Fanuc TP program (LS listing): UP025.LS

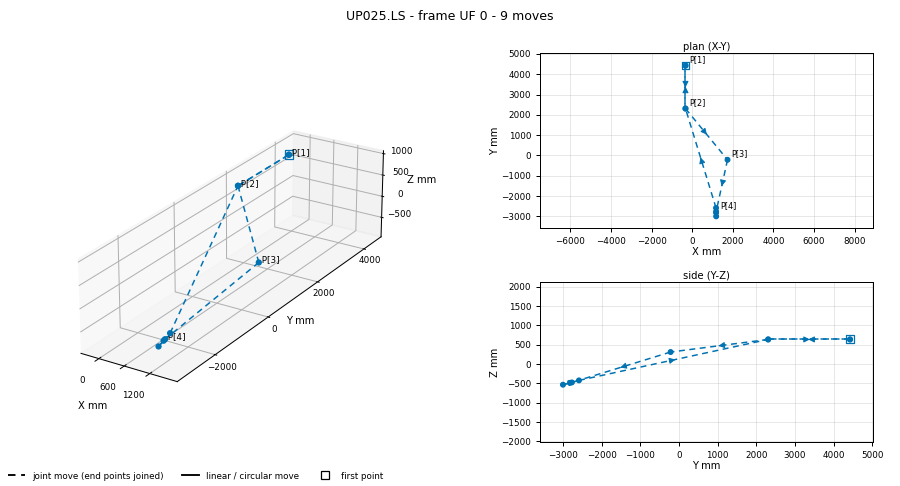
[picture p0: tool path of UP025.LS in frame UF 0, 9 of 9 moves have a stored position in this frame; points joined in program order, loops and branches not executed]
/PROG  UP025
/ATTR
OWNER		= MNEDITOR;
COMMENT		= "Int. 1680 Pos. 1";
PROG_SIZE	= 4392;
CREATE		= DATE 23-07-11  TIME 01:05:50;
MODIFIED	= DATE 24-07-27  TIME 15:01:24;
FILE_NAME	= UP005;
VERSION		= 0;
LINE_COUNT	= 18;
MEMORY_SIZE	= 7892;
PROTECT		= READ_WRITE;
TCD:  STACK_SIZE	= 500,
      TASK_PRIORITY	= 50,
      TIME_SLICE	= 0,
      BUSY_LAMP_OFF	= 0,
      ABORT_REQUEST	= 0,
      PAUSE_REQUEST	= 0;
DEFAULT_GROUP	= 1,1,1,1,*;
CONTROL_CODE	= 00000000 00000000;
/APPL
/MN
   1:  UFRAME_NUM=0 ;
   2:  UTOOL_NUM=1 ;
   3:  PAYLOAD[1] ;
   4:  !Apagar Perfil Lib. 77 vs ST1680 ;
   5:J P[1] 100% CNT0 ACC100 TB   0.00sec,P-SPS    ;
      1:  TC_ONLINE (ON) ;
      2:  DO[23]=OFF ;
      3:  TIMER[6]=RESET ;
      4:  TIMER[6]=START ;
      5:  CALL MAKRO050    ;
      6:  !Lib. de Herramientas ;
      7:  DO[80]=ON ;
      8:  DO[78]=OFF ;
      9:  DO[77]=ON ;
     10:  DO[75]=OFF ;
     11:  DO[74]=ON ;
     12:  DO[72]=OFF ;
     13:  !Lib. de Anticolisiones ;
     14:  DO[43]=ON ;
     15:  DO[44]=ON ;
     16:  !Apagar Pos. Base ;
     17:  DO[15]=OFF ;
     18:  !Robot en Trayectoria ;
     19:  DO[16]=ON ;
     20:  WAIT (!DI[61] AND DI[62] AND DI[77] AND M[2])    ;
     21:  DO[77]=OFF ;
     22:  WAIT (DI[23])    ;
     23:  DO[23]=ON ;
     24:  TC_ONLINE (!DI[61] AND DI[62] AND DI[77] AND M[2] AND M[30] AND M[31] AND M[33]) ;
       ------ ;
   6:J P[2] 100% CNT100 ACC100 TB   0.00sec,P-SPS    ;
      1:  TC_ONLINE (!DI[61] AND DI[62] AND DI[77] AND M[2] AND M[30] AND M[31] AND M[33]) ;
       ------ ;
   7:J P[3] 100% CNT100 ACC100 TB   0.00sec,P-SPS    ;
      1:  TC_ONLINE (!DI[61] AND DI[62] AND DI[77] AND M[2] AND M[30] AND M[31] AND M[33]) ;
       ------ ;
   8:J P[4] 100% CNT0 ACC100 TB    .10sec,P-SPS    ;
      1:  TC_ONLINE (ON) ;
      2:  DO[23]=OFF ;
      3:  F[2]=(ON) ;
      4:  CALL MAKRO343    ;
      5:  WAIT (M[34])    ;
      6:  WAIT (DI[23])    ;
      7:  DO[23]=ON ;
      8:  TC_ONLINE (DI[77] AND M[30] AND M[31] AND M[34]) ;
       ------ ;
   9:  !En Posicion ST1680-1 ;
  10:  !Tomar Pieza en ST1680-1 ;
  11:  !Fin de Trabajo 3 ;
  12:L P[5] 200mm/sec CNT0 ACC100 TB   0.00sec,P-SPS    ;
      1:  TC_ONLINE (ON) ;
      2:  DO[23]=OFF ;
      3:  DO[75]=ON ;
      4:  WAIT (M[1])    ;
      5:  F[2]=(ON) ;
      6:  CALL MAKRO342    ;
      7:  CALL MAKRO340    ;
      8:  WAIT (M[33])    ;
      9:  F[1]=(ON) ;
     10:  CALL MAKRO343    ;
     11:  WAIT (M[32])    ;
     12:  CALL MAKRO003    ;
     13:  GO[21]=2 ;
     14:  WAIT (DI[77])    ;
     15:  DO[75]=OFF ;
     16:  WAIT (DI[23])    ;
     17:  DO[23]=ON ;
     18:  TC_ONLINE (DI[77] AND M[30] AND M[32] AND M[33]) ;
       ------ ;
  13:  PAYLOAD[2] ;
  14:L P[6] 300mm/sec CNT0 ACC100 TB    .10sec,P-SPS    ;
      1:  TC_ONLINE (ON) ;
      2:  DO[23]=OFF ;
      3:  WAIT (DI[61] AND !DI[62])    ;
      4:  WAIT (DI[23])    ;
      5:  DO[23]=ON ;
      6:  TC_ONLINE (DI[61] AND !DI[62] AND DI[77] AND M[1] AND M[30] AND M[32] AND M[33]) ;
       ------ ;
  15:J P[7] 90% CNT100 ACC50 TB   0.00sec,P-SPS    ;
      1:  TC_ONLINE (DI[61] AND !DI[62] AND DI[77] AND M[1] AND M[30] AND M[32] AND M[33]) ;
       ------ ;
  16:J P[8] 90% CNT100 ACC75 TB   0.00sec,P-SPS    ;
      1:  TC_ONLINE (DI[61] AND !DI[62] AND DI[77] AND M[1] AND M[30] AND M[32] AND M[33]) ;
       ------ ;
  17:  !Encender Perfil Lib 77 vs ST1680 ;
  18:J P[9] 90% CNT0 ACC50 TB    .10sec,P-SPS    ;
      1:  TC_ONLINE (ON) ;
      2:  DO[23]=OFF ;
      3:  TIMER[6]=STOP ;
      4:  DO[77]=ON ;
      5:  WAIT (DI[23])    ;
      6:  DO[23]=ON ;
      7:  TC_ONLINE (M[1] AND M[30] AND M[32] AND M[33]) ;
       ------ ;
/POS
P[1]{
   GP1:
	UF : 0, UT : 1,		CONFIG : 'F U T, 0, 0, 0',
	X =  -332.978  mm,	Y =  4426.811  mm,	Z =   636.000  mm,
	W =    91.999 deg,	P =      .001 deg,	R =  -180.000 deg,
	E1=  2500.000  mm
   GP2:
	UF : 0, UT : 1,
	J1=     0.000  mm
   GP3:
	UF : 0, UT : 1,
	J1=     0.000  mm
   GP4:
	UF : 0, UT : 1,
	J1=     0.000  mm
};
P[2]{
   GP1:
	UF : 0, UT : 1,		CONFIG : 'F U T, 0, 0, 0',
	X =  -332.978  mm,	Y =  2308.572  mm,	Z =   636.000  mm,
	W =    91.999 deg,	P =     0.000 deg,	R =   180.000 deg,
	E1=   381.761  mm
   GP2:
	UF : 0, UT : 1,
	J1=     0.000  mm
   GP3:
	UF : 0, UT : 1,
	J1=     0.000  mm
   GP4:
	UF : 0, UT : 1,
	J1=     0.000  mm
};
P[3]{
   GP1:
	UF : 0, UT : 1,		CONFIG : 'F U T, 0, 0, 0',
	X =  1737.304  mm,	Y =  -214.852  mm,	Z =   310.171  mm,
	W =   -92.297 deg,	P =    29.499 deg,	R =   -87.049 deg,
	E1=   -31.039  mm
   GP2:
	UF : 0, UT : 1,
	J1=     0.000  mm
   GP3:
	UF : 0, UT : 1,
	J1=     0.000  mm
   GP4:
	UF : 0, UT : 1,
	J1=     0.000  mm
};
P[4]{
   GP1:
	UF : 0, UT : 1,		CONFIG : 'F U T, 0, 0, 0',
	X =  1175.296  mm,	Y = -2769.815  mm,	Z =  -476.333  mm,
	W =   -88.686 deg,	P =    14.319 deg,	R =   -89.512 deg,
	E1=   -67.734  mm
   GP2:
	UF : 0, UT : 1,
	J1=     0.000  mm
   GP3:
	UF : 0, UT : 1,
	J1=     0.000  mm
   GP4:
	UF : 0, UT : 1,
	J1=     0.000  mm
};
P[5]{
   GP1:
	UF : 0, UT : 1,		CONFIG : 'F U T, 0, 0, 0',
	X =  1177.251  mm,	Y = -2999.679  mm,	Z =  -535.012  mm,
	W =   -88.686 deg,	P =    14.320 deg,	R =   -89.512 deg,
	E1=   -67.734  mm
   GP2:
	UF : 0, UT : 1,
	J1=     0.000  mm
   GP3:
	UF : 0, UT : 1,
	J1=     0.000  mm
   GP4:
	UF : 0, UT : 1,
	J1=     0.000  mm
};
P[6]{
   GP1:
	UF : 0, UT : 1,		CONFIG : 'F U T, 0, 0, 0',
	X =  1174.699  mm,	Y = -2819.354  mm,	Z =  -487.291  mm,
	W =   -88.458 deg,	P =    14.512 deg,	R =   -89.509 deg,
	E1=   -67.734  mm
   GP2:
	UF : 0, UT : 1,
	J1=     0.000  mm
   GP3:
	UF : 0, UT : 1,
	J1=     0.000  mm
   GP4:
	UF : 0, UT : 1,
	J1=     0.000  mm
};
P[7]{
   GP1:
	UF : 0, UT : 1,		CONFIG : 'F U T, 0, 0, 0',
	X =  1172.046  mm,	Y = -2585.848  mm,	Z =  -423.241  mm,
	W =   -88.895 deg,	P =    14.619 deg,	R =   -89.503 deg,
	E1=   -67.735  mm
   GP2:
	UF : 0, UT : 1,
	J1=     0.000  mm
   GP3:
	UF : 0, UT : 1,
	J1=     0.000  mm
   GP4:
	UF : 0, UT : 1,
	J1=     0.000  mm
};
P[8]{
   GP1:
	UF : 0, UT : 1,		CONFIG : 'F U T, 0, 0, 0',
	X =  -332.978  mm,	Y =  2308.572  mm,	Z =   636.000  mm,
	W =    91.999 deg,	P =     0.000 deg,	R =  -180.000 deg,
	E1=   381.761  mm
   GP2:
	UF : 0, UT : 1,
	J1=     0.000  mm
   GP3:
	UF : 0, UT : 1,
	J1=     0.000  mm
   GP4:
	UF : 0, UT : 1,
	J1=     0.000  mm
};
P[9]{
   GP1:
	UF : 0, UT : 1,		CONFIG : 'F U T, 0, 0, 0',
	X =  -332.978  mm,	Y =  4426.811  mm,	Z =   636.000  mm,
	W =    91.999 deg,	P =      .001 deg,	R =  -180.000 deg,
	E1=  2500.000  mm
   GP2:
	UF : 0, UT : 1,
	J1=     0.000  mm
   GP3:
	UF : 0, UT : 1,
	J1=     0.000  mm
   GP4:
	UF : 0, UT : 1,
	J1=     0.000  mm
};
/END
